// TIA Portal V16 export
// export: Created 2023-03-29T11:03:30.6447831Z, ExportSetting WithDefaults, DisplayName Totally Integrated Automation Portal, DisplayVersion V16 Update 6, DisplayName TIA Portal Version Control Interface, DisplayVersion V16 Update 2, DisplayName TIA Portal Openness, DisplayVersion V16 Update 6, DisplayName STEP 7 Professional, DisplayVersion V16 Update 6, DisplayName STEP 7 Safety, DisplayVersion V16, DisplayName WinCC Advanced, DisplayVersion V16 Update 6
FUNCTION_BLOCK "alarm_petli-rtu_tcp"   // FB14, LAD
TITLE = kontrola obiegu pętli rtu, tcp
{ S7_Optimized_Access := 'TRUE' }
AUTHOR : rtecmer
VERSION : 0.1
// jeśli pętla się zawiesi bez sygnałizacji błędu w statusie to po ustalonym czasie 2x czas obiegu pętli nastąpi ustawienie znaczniku awaria pętli
// stored: AutoNumber true, IsIECCheckEnabled false, IsRetainMemResEnabled false, MemoryReserve 100, SetENOAutomatically false, UDAEnableTagReadback false
BEGIN

REGION Network 1: błąd petli Modbus TCP brak obiegu pętli
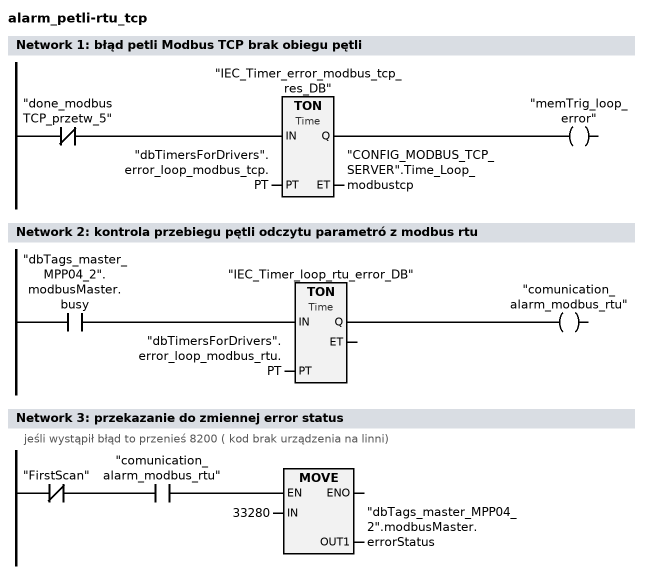
   RUNG wire#powerrail
      I_Contact( "done_modbusTCP_przetw_5" )
      { S7_Templates := "time_type := Time" } "IEC_Timer_error_modbus_tcp_res_DB".TON(pt := "dbTimersForDrivers".error_loop_modbus_tcp.PT, et => "CONFIG_MODBUS_TCP_SERVER".Time_Loop_modbustcp)
      Coil( "memTrig_loop_error" )
   END_RUNG
   // the same network as SCL:
   "IEC_Timer_error_modbus_tcp_res_DB".TON(IN := NOT "done_modbusTCP_przetw_5",
                           PT := "dbTimersForDrivers".error_loop_modbus_tcp.PT,
                           ET => "CONFIG_MODBUS_TCP_SERVER".Time_Loop_modbustcp);
   "memTrig_loop_error" := "IEC_Timer_error_modbus_tcp_res_DB".Q;
END_REGION

REGION Network 2: kontrola przebiegu pętli odczytu parametró z modbus rtu
   RUNG wire#powerrail
      Contact( "dbTags_master_MPP04_2".modbusMaster.busy )
      { S7_Templates := "time_type := Time" } "IEC_Timer_loop_rtu_error_DB".TON(pt := "dbTimersForDrivers".error_loop_modbus_rtu.PT, et =>)
      Coil( "comunication_alarm_modbus_rtu" )
   END_RUNG
   // the same network as SCL:
   "IEC_Timer_loop_rtu_error_DB".TON(IN := "dbTags_master_MPP04_2".modbusMaster.busy,
                           PT := "dbTimersForDrivers".error_loop_modbus_rtu.PT);
   "comunication_alarm_modbus_rtu" := "IEC_Timer_loop_rtu_error_DB".Q;
END_REGION

REGION Network 3: przekazanie do zmiennej error status
   // jeśli wystąpił błąd to przenieś 8200 ( kod brak urządzenia na linni)
   RUNG wire#powerrail
      I_Contact( "FirstScan" )
      Contact( "comunication_alarm_modbus_rtu" )
      Move(in := 33280, out1 => "dbTags_master_MPP04_2".modbusMaster.errorStatus)
   END_RUNG
   // the same network as SCL:
   IF NOT "FirstScan" AND "comunication_alarm_modbus_rtu" THEN
       "dbTags_master_MPP04_2".modbusMaster.errorStatus := 33280;
   END_IF;
END_REGION
END_FUNCTION_BLOCK
